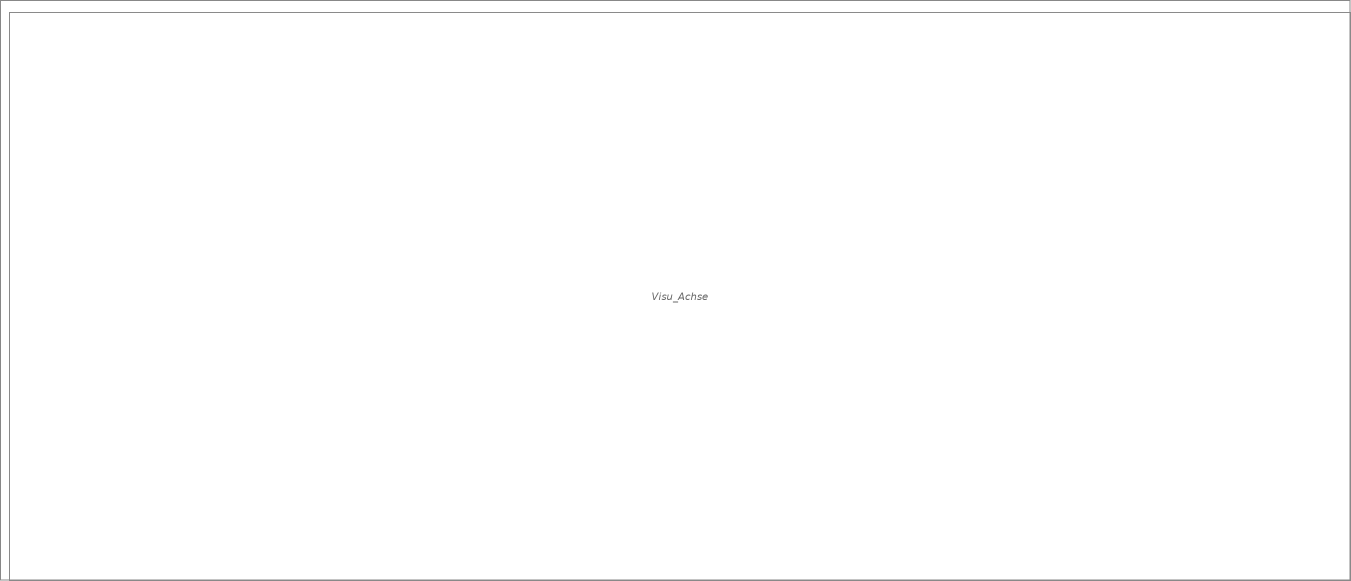
VISUALIZATION Achse_S  // 1351x581
    Frame (9,12 1342x569)
        shows Visu_Achse(Axis := MAIN.Axis_S)
END_VISUALIZATION

(* stored: Version 1.1.0.1, ProductVersion 3.1.4024.10
   Visu Achse_S: Id {60f747f0-89c5-43ea-9f8c-2d297b4ebc67} *)
